Universal Robots PolyScope program: ghTest202408061747.urp

Program ghTest202408061747 (installation=cube_dev1 directory=/programs createdIn=5.11.11.0 lastSavedIn=5.11.5.1010327 robotSerialNumber=20215500677)
Calibrated DH parameters: a=[0.000204, -0.239222, -0.391845, -0.000001, 0.000022, 0]; d=[0.162722, -355.808559, 353.37206, 2.570385, 0.099741, 0.099629]; alpha=[1.571124, 0.000988, 0.008295, 1.568963, -1.570303, 0]; deltaTheta=[0, -0.973091, 7.204745, 0.05153, 0, 0]
Robot Program (runOnlyOnce=true)
  Script file ghTest202408061747.script
    | def Program():
    |   DefaultGHToolTcp = p[-0.108, 0.063, 0.084, -0.61394, 0.61394, 1.48219]
    |   DefaultGHToolWeight = 0
    |   DefaultGHToolCog = [-0.108, 0.063, 0.084]
    |   DefaultSpeed = 0.1
    |   DefaultZone = 0
    |   Wait000 = 2
    |   set_tcp(DefaultGHToolTcp)
    |   set_payload(DefaultGHToolWeight, DefaultGHToolCog)
    |   movej([2.1642, -2.4609, 2.4609, 2.81, -1.0297, 0.0524], a=3.1416, v=0.3142, r=DefaultZone)
    |   movej([0.784, -0.0272, 4.9749, 3.5225, -2.0936, 2.5275], a=3.1416, v=0.2537, r=DefaultZone)
    |   set_digital_out(1,True)
    |   sleep(Wait000)
    |   force_mode(p[0.466762,-0.259202,0.632648,0,2.356194,0], [0,0,1,0,0,0], [0,0,5,0,0,0], 2, [.1,.1,0.05,.785,.785,.785])
    |   movej([-0.4135, -0.076, 4.3255, 4.3459, -1.2827, 3.4424], a=3.1416, v=0.218, r=DefaultZone)
    |   set_digital_out(1,True)
    |   sleep(Wait000)
    |   force_mode(p[0.466762,-0.259202,0.632648,0,2.356194,0], [0,0,1,0,0,0], [0,0,5,0,0,0], 2, [.1,.1,0.05,.785,.785,.785])
    |   movej([1.7938, -0.3514, 4.4756, 3.5122, -2.3317, 1.2605], a=3.1416, v=0.3928, r=DefaultZone)
    |   set_digital_out(1,True)
    |   sleep(Wait000)
    |   force_mode(p[0.466762,-0.259202,0.632648,0,2.356194,0], [0,0,1,0,0,0], [0,0,5,0,0,0], 2, [.1,.1,0.05,.785,.785,.785])
    |   movej([1.6083, -0.1713, 5.1097, 2.8782, -2.3555, 1.5178], a=3.1416, v=0.1154, r=DefaultZone)
    |   set_digital_out(1,True)
    |   sleep(Wait000)
    |   force_mode(p[0.466762,-0.259202,0.632648,0,2.356194,0], [0,0,1,0,0,0], [0,0,5,0,0,0], 2, [.1,.1,0.05,.785,.785,.785])
    |   movej([0.784, -0.0272, 4.9749, 3.5225, -2.0936, 2.5275], a=3.1416, v=0.1797, r=DefaultZone)
    |   set_digital_out(1,True)
    |   sleep(Wait000)
    |   force_mode(p[0.466762,-0.259202,0.632648,0,2.356194,0], [0,0,1,0,0,0], [0,0,5,0,0,0], 2, [.1,.1,0.05,.785,.785,.785])
    |   movej([2.1642, -2.4609, 2.4609, 2.81, -1.0297, 0.0524], a=3.1416, v=0.3179, r=DefaultZone)
    |   movej([0.784, -0.0272, 4.9749, 3.5225, -2.0936, 2.5275], a=3.1416, v=0.2537, r=DefaultZone)
    |   set_digital_out(1,True)
    |   sleep(Wait000)
    |   force_mode(p[0.466762,0.105798,0.632648,-0.729011,1.759988,-1.759988], [0,0,1,0,0,0], [0,0,5,0,0,0], 2, [.1,.1,0.05,.785,.785,.785])
    |   movej([-0.4135, -0.076, 4.3255, 4.3459, -1.2827, 3.4424], a=3.1416, v=0.218, r=DefaultZone)
    |   set_digital_out(1,True)
    |   sleep(Wait000)
    |   force_mode(p[0.466762,0.105798,0.632648,-0.729011,1.759988,-1.759988], [0,0,1,0,0,0], [0,0,5,0,0,0], 2, [.1,.1,0.05,.785,.785,.785])
    |   movej([1.7938, -0.3514, 4.4756, 3.5122, -2.3317, 1.2605], a=3.1416, v=0.3928, r=DefaultZone)
    |   set_digital_out(1,True)
    |   sleep(Wait000)
    |   force_mode(p[0.466762,0.105798,0.632648,-0.729011,1.759988,-1.759988], [0,0,1,0,0,0], [0,0,5,0,0,0], 2, [.1,.1,0.05,.785,.785,.785])
    |   movej([1.6083, -0.1713, 5.1097, 2.8782, -2.3555, 1.5178], a=3.1416, v=0.1154, r=DefaultZone)
    |   set_digital_out(1,True)
    |   sleep(Wait000)
    |   force_mode(p[0.466762,0.105798,0.632648,-0.729011,1.759988,-1.759988], [0,0,1,0,0,0], [0,0,5,0,0,0], 2, [.1,.1,0.05,.785,.785,.785])
    |   movej([0.784, -0.0272, 4.9749, 3.5225, -2.0936, 2.5275], a=3.1416, v=0.1797, r=DefaultZone)
    |   set_digital_out(1,True)
    |   sleep(Wait000)
    |   force_mode(p[0.466762,0.105798,0.632648,-0.729011,1.759988,-1.759988], [0,0,1,0,0,0], [0,0,5,0,0,0], 2, [.1,.1,0.05,.785,.785,.785])
    |   movej([2.1642, -2.4609, 2.4609, 2.81, -1.0297, 0.0524], a=3.1416, v=0.3179, r=DefaultZone)
    |   movej([0.784, -0.0272, 4.9749, 3.5225, -2.0936, 2.5275], a=3.1416, v=0.2537, r=DefaultZone)
    |   set_digital_out(1,True)
    |   sleep(Wait000)
    |   force_mode(p[0.466762,0.105798,0.267648,1.202235,0,2.902453], [0,0,1,0,0,0], [0,0,5,0,0,0], 2, [.1,.1,0.05,.785,.785,.785])
    |   movej([-0.4135, -0.076, 4.3255, 4.3459, -1.2827, 3.4424], a=3.1416, v=0.218, r=DefaultZone)
    |   set_digital_out(1,True)
    |   sleep(Wait000)
    |   force_mode(p[0.466762,0.105798,0.267648,1.202235,0,2.902453], [0,0,1,0,0,0], [0,0,5,0,0,0], 2, [.1,.1,0.05,.785,.785,.785])
    |   movej([1.7938, -0.3514, 4.4756, 3.5122, -2.3317, 1.2605], a=3.1416, v=0.3928, r=DefaultZone)
    |   set_digital_out(1,True)
    |   sleep(Wait000)
    |   force_mode(p[0.466762,0.105798,0.267648,1.202235,0,2.902453], [0,0,1,0,0,0], [0,0,5,0,0,0], 2, [.1,.1,0.05,.785,.785,.785])
    |   movej([1.6083, -0.1713, 5.1097, 2.8782, -2.3555, 1.5178], a=3.1416, v=0.1154, r=DefaultZone)
    |   set_digital_out(1,True)
    |   sleep(Wait000)
    |   force_mode(p[0.466762,0.105798,0.267648,1.202235,0,2.902453], [0,0,1,0,0,0], [0,0,5,0,0,0], 2, [.1,.1,0.05,.785,.785,.785])
    |   movej([0.784, -0.0272, 4.9749, 3.5225, -2.0936, 2.5275], a=3.1416, v=0.1797, r=DefaultZone)
    |   set_digital_out(1,True)
    |   sleep(Wait000)
    |   force_mode(p[0.466762,0.105798,0.267648,1.202235,0,2.902453], [0,0,1,0,0,0], [0,0,5,0,0,0], 2, [.1,.1,0.05,.785,.785,.785])
    |   movej([2.1642, -2.4609, 2.4609, 2.81, -1.0297, 0.0524], a=3.1416, v=0.3179, r=DefaultZone)
    |   movej([0.784, -0.0272, 4.9749, 3.5225, -2.0936, 2.5275], a=3.1416, v=0.2537, r=DefaultZone)
    |   set_digital_out(1,True)
    |   sleep(Wait000)
    |   force_mode(p[0.466762,-0.259202,0.267648,0.729011,1.759988,1.759988], [0,0,1,0,0,0], [0,0,5,0,0,0], 2, [.1,.1,0.05,.785,.785,.785])
    |   movej([-0.4135, -0.076, 4.3255, 4.3459, -1.2827, 3.4424], a=3.1416, v=0.218, r=DefaultZone)
    |   set_digital_out(1,True)
    |   sleep(Wait000)
    |   force_mode(p[0.466762,-0.259202,0.267648,0.729011,1.759988,1.759988], [0,0,1,0,0,0], [0,0,5,0,0,0], 2, [.1,.1,0.05,.785,.785,.785])
    |   movej([1.7938, -0.3514, 4.4756, 3.5122, -2.3317, 1.2605], a=3.1416, v=0.3928, r=DefaultZone)
    |   set_digital_out(1,True)
    |   sleep(Wait000)
    |   force_mode(p[0.466762,-0.259202,0.267648,0.729011,1.759988,1.759988], [0,0,1,0,0,0], [0,0,5,0,0,0], 2, [.1,.1,0.05,.785,.785,.785])
    |   movej([1.6083, -0.1713, 5.1097, 2.8782, -2.3555, 1.5178], a=3.1416, v=0.1154, r=DefaultZone)
    |   set_digital_out(1,True)
    |   sleep(Wait000)
    |   force_mode(p[0.466762,-0.259202,0.267648,0.729011,1.759988,1.759988], [0,0,1,0,0,0], [0,0,5,0,0,0], 2, [.1,.1,0.05,.785,.785,.785])
    |   movej([0.784, -0.0272, 4.9749, 3.5225, -2.0936, 2.5275], a=3.1416, v=0.1797, r=DefaultZone)
    |   set_digital_out(1,True)
    |   sleep(Wait000)
    |   force_mode(p[0.466762,-0.259202,0.267648,0.729011,1.759988,1.759988], [0,0,1,0,0,0], [0,0,5,0,0,0], 2, [.1,.1,0.05,.785,.785,.785])
    | end
    | Program()
